{attribute 'qualified_only'}
{attribute 'to_string'}
TYPE E_LinearActuatorStates :
(
	Idle:=0,
	Resetting,
	Homing1,
	Homing2,
	Disabled,
	Enabled,
	Jogging,
	MovingAbs,
	Halting
)UINT := Idle
;
END_TYPE

(* stored: Version 1.1.0.1, ProductVersion 3.1.4024.12
   EnumerationTextList E_LinearActuatorStates: Id {387a57e9-e3bd-4ea5-a059-ff3417d4364a} *)
